(* Logix 5000 project; controller Ex_2_17 Emulate 5570 rev 33.11; software revision 33.00 *)
// Palletizibg jerrycans with a robot

TASK MainTask (continuous, watchdog 500 ms) : MainProgram

MODULES
   Local : Emulate 5570 (ICP 4, rev 33.11)
END_MODULES

VAR_GLOBAL   (* controller tags *)
   B1 : BOOL;   // Sensor B1
   B2 : BOOL;   // Sensor B2
   B3 : BOOL;   // Sensor B3
   M1 : BOOL;   // Motor M1
   M3_DI : BOOL;   // DI_Robot Controller
   M3_DO : BOOL;
   P1 : BOOL;   // Lamp P1
   Robot_Ready : BOOL;
END_VAR

PROGRAM MainProgram   (* main routine MainRoutine *)

ROUTINE MainRoutine   (* ladder *)
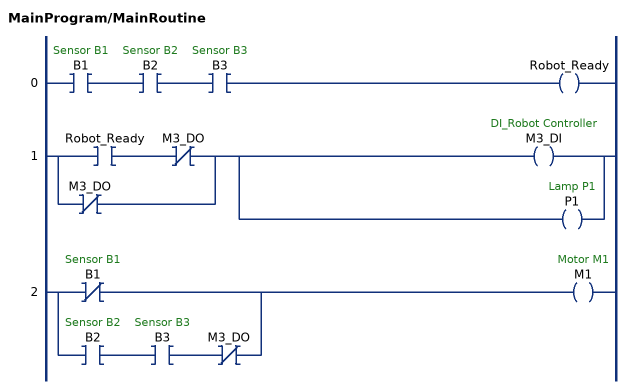
   0: XIC(B1)XIC(B2)XIC(B3)OTE(Robot_Ready);
   1: [XIC(Robot_Ready) XIO(M3_DO) ,XIO(M3_DO) ][OTE(M3_DI) ,OTE(P1) ];
   2: [XIO(B1) ,XIC(B2) XIC(B3) XIO(M3_DO) ]OTE(M1);
END_ROUTINE
END_PROGRAM
